// TwinCAT 3 PLC project OSCATTests
// ProgramVersion: 3.1.4023.0
// libraries:
//   OSCAT, * (RWTH Aachen University - E.ON Energy Research Center)
//   Tc2_Standard, * (Beckhoff Automation GmbH)
//   Tc2_System, * (Beckhoff Automation GmbH)
//   Tc3_Module, * (Beckhoff Automation GmbH)
//   TcUnit, * (www.tcunit.org)
// project tree:
//   oscat_basic/Engineering/signal processing/ FILTER_MAV_DW_Test.TcPOU, FILTER_MAV_W_Test.TcPOU
//   oscat_basic/Mathematical/ FLOOR_Test.TcPOU
//   / PlcTask.TcTTO, PRG_TEST.TcPOU
//   POUs/ MAIN.TcPOU
// real-time tasks:
//   TASK PlcTask: cycle T#10ms, priority 20, ADS port 350

CONFIGURATION OSCATTests
    RESOURCE PLC ON TwinCAT3
        TASK PlcTask(INTERVAL := T#10ms, PRIORITY := 20);
        PROGRAM PRG_TEST WITH PlcTask : PRG_TEST;
    END_RESOURCE
END_CONFIGURATION

// ---- PRG_TEST.TcPOU
PROGRAM PRG_TEST
VAR
	fbFLOOR_Test : FLOOR_Test;
	fbMAV_DW_Test : FILTER_MAV_DW_Test; 
	//fbMAV_W_Test : FILTER_MAV_W_Test; 
END_VAR

TcUnit.RUN();

END_PROGRAM

// ---- oscat_basic/Mathematical/FLOOR_Test.TcPOU
FUNCTION_BLOCK FLOOR_Test EXTENDS FB_TestSuite
VAR_INPUT
END_VAR
VAR_OUTPUT
END_VAR
VAR
END_VAR

PositivePieToThree();
NegativePieToNegativeFour();
TwoToTwo();

METHOD NegativePieToNegativeFour
VAR
	Result : INT;
	ExpectedFloor : INT := -4;
END_VAR
TEST('NegativePieToNegativeFour');
 
Result := FLOOR(X := -3.14);
 
AssertEquals(Expected := ExpectedFloor,
             Actual := Result,
             Message := 'The calculation is not correct');
 
TEST_FINISHED();
END_METHOD

METHOD PositivePieToThree
VAR
	Result : INT;
	ExpectedFloor : INT := 3; 
END_VAR
TEST('PositivePieToThree');
 
Result := FLOOR(X := 3.14);
 
AssertEquals(Expected := ExpectedFloor,
             Actual := Result,
             Message := 'The calculation is not correct');
 
TEST_FINISHED();
END_METHOD

METHOD TwoToTwo
VAR
	Result : INT;
	ExpectedFloor : INT := 2;
END_VAR
TEST('TwoToTwo');
 
Result := FLOOR(X := 2);
 
AssertEquals(Expected := ExpectedFloor,
             Actual := Result,
             Message := 'The calculation is not correct');
 
TEST_FINISHED();
END_METHOD

END_FUNCTION_BLOCK

// ---- oscat_basic/Engineering/signal processing/FILTER_MAV_DW_Test.TcPOU
FUNCTION_BLOCK FILTER_MAV_DW_Test EXTENDS FB_TestSuite
VAR_INPUT
END_VAR
VAR_OUTPUT
END_VAR
VAR
END_VAR

AverageEightThenTenEqualsNine();
AverageTenThenEightEqualsNine();

METHOD AverageEightThenTenEqualsNine
VAR
	MAV : FILTER_MAV_DW;
	Result : DWORD;
	ExpectedAverage : DWORD := 9;
END_VAR
TEST('AverageEightThenTenEqualsNine');
 
MAV(X := 8, N := 2);
MAV(X := 10, Y => Result);
 
AssertEquals(Expected := ExpectedAverage,
             Actual := Result,
             Message := 'The calculation is not correct');
 
TEST_FINISHED();
END_METHOD

METHOD AverageTenThenEightEqualsNine
VAR
	MAV : FILTER_MAV_DW;
	Result : DWORD;
	ExpectedAverage : DWORD := 9;
END_VAR
TEST('AverageTenThenEightEqualsNine');
 
MAV(X := 10, N := 2);
MAV(X := 8, Y => Result);
 
AssertEquals(Expected := ExpectedAverage,
             Actual := Result,
             Message := 'The calculation is not correct');
 
TEST_FINISHED();
END_METHOD

END_FUNCTION_BLOCK

// ---- oscat_basic/Engineering/signal processing/FILTER_MAV_W_Test.TcPOU
FUNCTION_BLOCK FILTER_MAV_W_Test EXTENDS FB_TestSuite
VAR_INPUT
END_VAR
VAR_OUTPUT
END_VAR
VAR
END_VAR

AverageEightThenTenEqualsNine();
AverageTenThenEightEqualsNine();

METHOD AverageEightThenTenEqualsNine
VAR
	MAV : FILTER_MAV_W;
	Result : WORD;
	ExpectedAverage : WORD := 9;
END_VAR
TEST('AverageEightThenTenEqualsNine');
 
MAV(X := 8, N := 2);
MAV(X := 10, Y => Result);
 
AssertEquals(Expected := ExpectedAverage,
             Actual := Result,
             Message := 'The calculation is not correct');
 
TEST_FINISHED();
END_METHOD

METHOD AverageTenThenEightEqualsNine
VAR
	MAV : FILTER_MAV_W;
	Result : WORD;
	ExpectedAverage : WORD := 9;
END_VAR
TEST('AverageTenThenEightEqualsNine');
 
MAV(X := 10, N := 2);
MAV(X := 8, Y => Result);
 
AssertEquals(Expected := ExpectedAverage,
             Actual := Result,
             Message := 'The calculation is not correct');
 
TEST_FINISHED();
END_METHOD

END_FUNCTION_BLOCK

// ---- POUs/MAIN.TcPOU
PROGRAM MAIN
VAR
END_VAR

END_PROGRAM
